// TIA Portal V19 export
TYPE "TAx_Pos_Sts"
// stored: Access Published
   STRUCT
      AlarmPresence : Bool;   // Cumulative alarm presence
      WarningPresence : Bool;   // Cumulative warning presence
      Enabled : Bool;   // Axis is enabled
      Done : Bool;
      Standstill : Bool;   // Axis is standstill
      RstHWDone : Bool;   // Reset hardware done
      Homed : Bool;
      AtProgrammedSpeed : Bool;
      HomingPermitted : Bool;
      HomingDone : Bool;
      MoveMinusPermitted : Bool;
      MovePlusPermitted : Bool;
      MoveAbsPermitted : Bool;
      Positioned : Bool;
      ActualPosition : LReal;
      ActualSpeed : LReal;
      ActualTarget : LReal;
      SwLimitPlus : LReal;
      SwLimitMinus : LReal;
   END_STRUCT;
END_TYPE
